{attribute 'GeneratedUsingTerminal: EL9930-0000-0016'}
{attribute addProperty BoxType "EL9930-0000-0016"}
{attribute addProperty Description "EL9930-0000, PROFIsafe-Segment-Abschlussklemme Primary"}
{attribute addProperty Physics "KKK"}
{attribute addProperty Id "IO_InputsEMPTY_STRUCTURE0IO_OutputsEMPTY_STRUCTURE0WcStateAT %I*WcState_9091E0EB2InfoDataAT %I*InfoData_90184F0C16"}
{attribute addProperty CRC "2007939653"}
{attribute addProperty Size "18"}
TYPE EL9930_77AEBA45 EXTENDS EtcSlaveTerminalBase_947E5A46 :
STRUCT
	{attribute addProperty Name "IO_Inputs"}
	IO_Inputs : EMPTY_STRUCTURE;
	{attribute addProperty Name "IO_Outputs"}
	IO_Outputs : EMPTY_STRUCTURE;
	{attribute addProperty Name "WcState"}
	WcState : WcState_9091E0EB;
	{attribute addProperty Name "InfoData"}
	InfoData : InfoData_90184F0C;
END_STRUCT
END_TYPE

(* stored: Version 1.2.0.0, ProductVersion 3.1.4024.9
   DUT EL9930_77AEBA45: Id {71d413f6-6004-47b2-934e-38f1c1886b15} *)
